// TIA Portal V21 export
FUNCTION "FC601" : Void   // FC601, LAD
TITLE = FC601
{ S7_Optimized_Access := 'TRUE' }
// MAIN CIP CALL BLOCK
// stored: AutoNumber false, SetENOAutomatically false
   VAR_TEMP   // added for the SCL form of the ladder/FBD networks
      _w1 : Bool;
      _w2 : Bool;
      _w3 : Bool;
   END_VAR
BEGIN

REGION Network 1: "FC604"
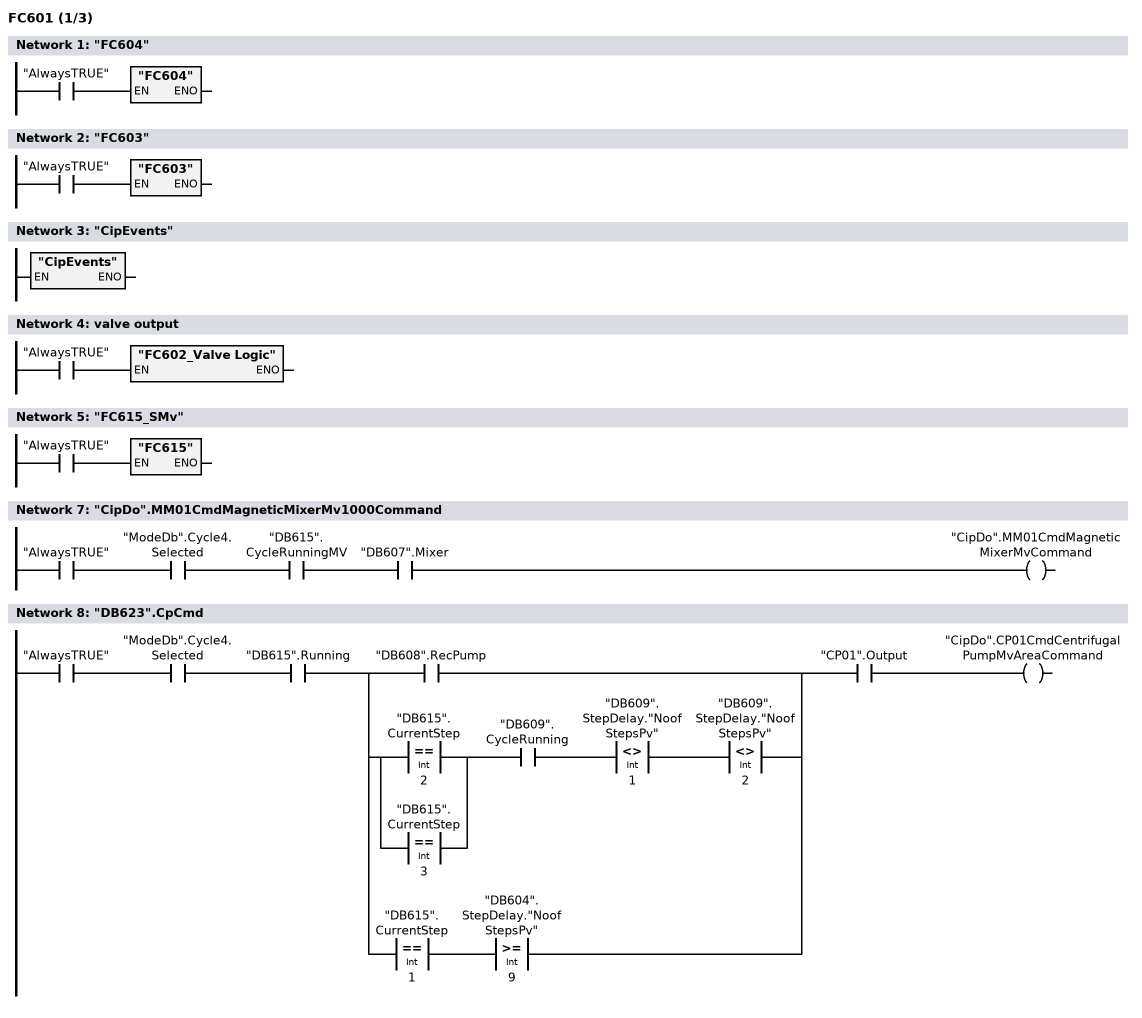
   RUNG wire#powerrail
      Contact( "AlwaysTRUE" )
      "FC604"()
   END_RUNG
   // the same network as SCL:
   IF "AlwaysTRUE" THEN "FC604"(); END_IF;
END_REGION

REGION Network 2: "FC603"
   RUNG wire#powerrail
      Contact( "AlwaysTRUE" )
      "FC603"()
   END_RUNG
   // the same network as SCL:
   IF "AlwaysTRUE" THEN "FC603"(); END_IF;
END_REGION

REGION Network 3: "CipEvents"
   RUNG wire#powerrail
      "CipEvents"()
   END_RUNG
   // the same network as SCL:
   "CipEvents"();
END_REGION

REGION Network 4: valve output
   RUNG wire#powerrail
      Contact( "AlwaysTRUE" )
      "FC602_Valve Logic"()
   END_RUNG
   // the same network as SCL:
   IF "AlwaysTRUE" THEN "FC602_Valve Logic"(); END_IF;
END_REGION

REGION Network 5: "FC615_SMv"
   RUNG wire#powerrail
      Contact( "AlwaysTRUE" )
      "FC615"()
   END_RUNG
   // the same network as SCL:
   IF "AlwaysTRUE" THEN "FC615"(); END_IF;
END_REGION

REGION Network 6: *************DO ***********************
END_REGION

REGION Network 7: "CipDo".MM01CmdMagneticMixerMv1000Command
   RUNG wire#powerrail
      Contact( "AlwaysTRUE" )
      Contact( "ModeDb".Cycle4.Selected )
      Contact( "DB615".CycleRunningMV )
      Contact( "DB607".Mixer )
      Coil( "CipDo".MM01CmdMagneticMixerMvCommand )
   END_RUNG
   // the same network as SCL:
   "CipDo".MM01CmdMagneticMixerMvCommand := "AlwaysTRUE" AND "ModeDb".Cycle4.Selected AND "DB615".CycleRunningMV AND "DB607".Mixer;
END_REGION

REGION Network 8: "DB623".CpCmd
   RUNG wire#powerrail
      Contact( "AlwaysTRUE" )
      Contact( "ModeDb".Cycle4.Selected )
      Contact( "DB615".Running )
      wire#w1
      Contact( "DB608".RecPump )
      wire#w2
      Contact( "CP01".Output )
      Coil( "CipDo".CP01CmdCentrifugalPumpMvAreaCommand )
   END_RUNG
   RUNG wire#w1
      { S7_Templates := "SrcType := Int" } EQ_Contact(in1 := "DB615".CurrentStep, in2 := 2)
      wire#w3
      Contact( "DB609".CycleRunning )
      { S7_Templates := "SrcType := Int" } NE_Contact(in1 := "DB609".StepDelay."Noof StepsPv", in2 := 1)
      { S7_Templates := "SrcType := Int" } NE_Contact(in1 := "DB609".StepDelay."Noof StepsPv", in2 := 2)
   END_RUNG wire#w2
   RUNG wire#w1
      { S7_Templates := "SrcType := Int" } EQ_Contact(in1 := "DB615".CurrentStep, in2 := 3)
   END_RUNG wire#w3
   RUNG wire#w1
      { S7_Templates := "SrcType := Int" } EQ_Contact(in1 := "DB615".CurrentStep, in2 := 1)
      { S7_Templates := "SrcType := Int" } GE_Contact(in1 := "DB604".StepDelay."Noof StepsPv", in2 := 9)
   END_RUNG wire#w2
   // the same network as SCL:
   "CipDo".CP01CmdCentrifugalPumpMvAreaCommand := "AlwaysTRUE" AND "ModeDb".Cycle4.Selected AND "DB615".Running AND ("DB608".RecPump OR ((("DB615".CurrentStep = 2) OR ("DB615".CurrentStep = 3)) AND "DB609".CycleRunning AND ("DB609".StepDelay."Noof StepsPv" <> 1) AND ("DB609".StepDelay."Noof StepsPv" <> 2)) OR (("DB615".CurrentStep = 1) AND ("DB604".StepDelay."Noof StepsPv" >= 9))) AND "CP01".Output;
END_REGION

REGION Network 9: "CipDo".CP01CmdCentrifugalPump
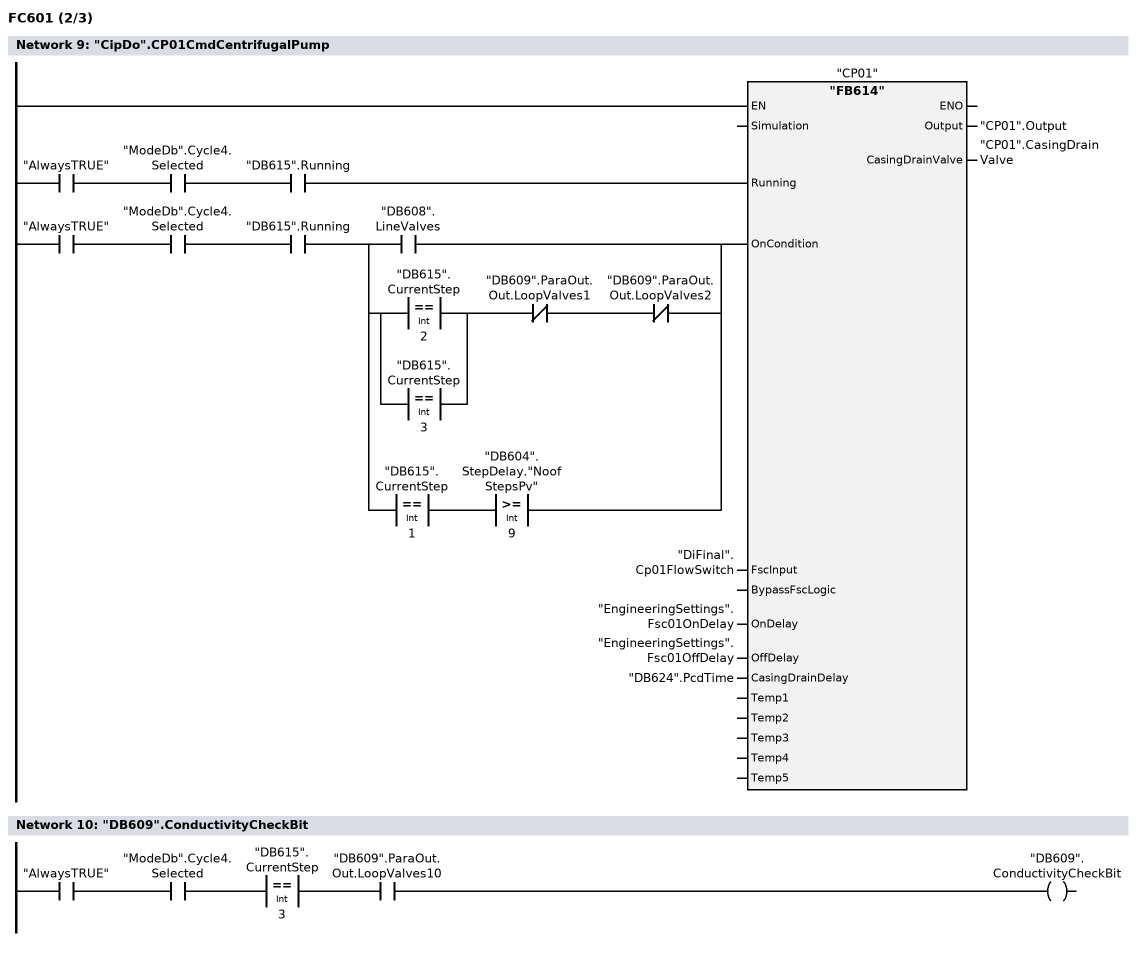
   RUNG wire#powerrail
      "CP01"(Running := wire#w1, OnCondition := wire#w4, Simulation :=, FscInput := "DiFinal".Cp01FlowSwitch, BypassFscLogic :=, OnDelay := "EngineeringSettings".Fsc01OnDelay, OffDelay := "EngineeringSettings".Fsc01OffDelay, CasingDrainDelay := "DB624".PcdTime, Temp1 :=, Temp2 :=, Temp3 :=, Temp4 :=, Temp5 :=, Output => "CP01".Output, CasingDrainValve => "CP01".CasingDrainValve)
   END_RUNG
   RUNG wire#powerrail
      Contact( "AlwaysTRUE" )
      Contact( "ModeDb".Cycle4.Selected )
      Contact( "DB615".Running )
   END_RUNG wire#w1
   RUNG wire#powerrail
      Contact( "AlwaysTRUE" )
      Contact( "ModeDb".Cycle4.Selected )
      Contact( "DB615".Running )
      wire#w2
      Contact( "DB608".LineValves )
   END_RUNG wire#w4
   RUNG wire#w2
      { S7_Templates := "SrcType := Int" } EQ_Contact(in1 := "DB615".CurrentStep, in2 := 2)
      wire#w3
      I_Contact( "DB609".ParaOut.Out.LoopValves1 )
      I_Contact( "DB609".ParaOut.Out.LoopValves2 )
   END_RUNG wire#w4
   RUNG wire#w2
      { S7_Templates := "SrcType := Int" } EQ_Contact(in1 := "DB615".CurrentStep, in2 := 3)
   END_RUNG wire#w3
   RUNG wire#w2
      { S7_Templates := "SrcType := Int" } EQ_Contact(in1 := "DB615".CurrentStep, in2 := 1)
      { S7_Templates := "SrcType := Int" } GE_Contact(in1 := "DB604".StepDelay."Noof StepsPv", in2 := 9)
   END_RUNG wire#w4
   // the same network as SCL:
   "CP01"(Running := "AlwaysTRUE" AND "ModeDb".Cycle4.Selected AND "DB615".Running,   // "FB614"
          OnCondition := "AlwaysTRUE" AND "ModeDb".Cycle4.Selected AND "DB615".Running AND ("DB608".LineValves OR ((("DB615".CurrentStep = 2) OR ("DB615".CurrentStep = 3)) AND NOT "DB609".ParaOut.Out.LoopValves1 AND NOT "DB609".ParaOut.Out.LoopValves2) OR (("DB615".CurrentStep = 1) AND ("DB604".StepDelay."Noof StepsPv" >= 9))),
          FscInput := "DiFinal".Cp01FlowSwitch,
          OnDelay := "EngineeringSettings".Fsc01OnDelay,
          OffDelay := "EngineeringSettings".Fsc01OffDelay,
          CasingDrainDelay := "DB624".PcdTime,
          Output => "CP01".Output,
          CasingDrainValve => "CP01".CasingDrainValve);
END_REGION

REGION Network 10: "DB609".ConductivityCheckBit
   RUNG wire#powerrail
      Contact( "AlwaysTRUE" )
      Contact( "ModeDb".Cycle4.Selected )
      { S7_Templates := "SrcType := Int" } EQ_Contact(in1 := "DB615".CurrentStep, in2 := 3)
      Contact( "DB609".ParaOut.Out.LoopValves10 )
      Coil( "DB609".ConductivityCheckBit )
   END_RUNG
   // the same network as SCL:
   "DB609".ConductivityCheckBit := "AlwaysTRUE" AND "ModeDb".Cycle4.Selected AND ("DB615".CurrentStep = 3) AND "DB609".ParaOut.Out.LoopValves10;
END_REGION

REGION Network 12: "ProcessAlarms".MvVesselWfiFlowLow
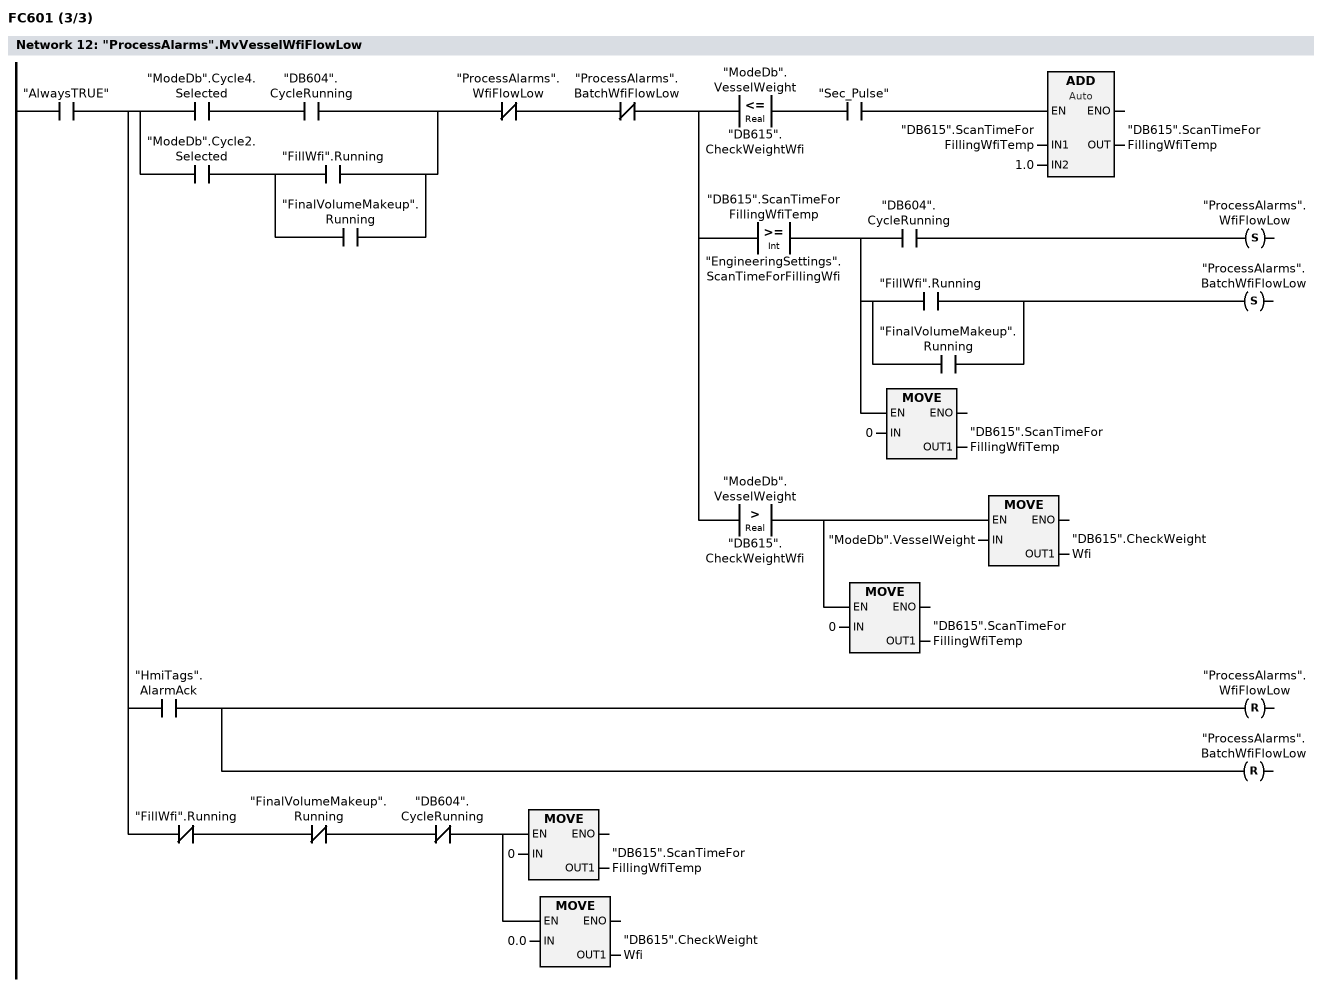
   RUNG wire#powerrail
      Contact( "AlwaysTRUE" )
      wire#w1
      Contact( "ModeDb".Cycle4.Selected )
      Contact( "DB604".CycleRunning )
      wire#w2
      I_Contact( "ProcessAlarms".WfiFlowLow )
      I_Contact( "ProcessAlarms".BatchWfiFlowLow )
      wire#w4
      { S7_Templates := "SrcType := Real" } LE_Contact(in1 := "ModeDb".VesselWeight, in2 := "DB615".CheckWeightWfi)
      Contact( "Sec_Pulse" )
      Add(in1 := "DB615".ScanTimeForFillingWfiTemp, in2 := 1.0, out => "DB615".ScanTimeForFillingWfiTemp)
   END_RUNG
   RUNG wire#w1
      Contact( "ModeDb".Cycle2.Selected )
      wire#w3
      Contact( "FillWfi".Running )
   END_RUNG wire#w2
   RUNG wire#w3
      Contact( "FinalVolumeMakeup".Running )
   END_RUNG wire#w2
   RUNG wire#w4
      { S7_Templates := "SrcType := Int" } GE_Contact(in1 := "DB615".ScanTimeForFillingWfiTemp, in2 := "EngineeringSettings".ScanTimeForFillingWfi)
      wire#w5
      Contact( "DB604".CycleRunning )
      S_Coil( "ProcessAlarms".WfiFlowLow )
   END_RUNG
   RUNG wire#w5
      Contact( "FillWfi".Running )
      wire#w6
      S_Coil( "ProcessAlarms".BatchWfiFlowLow )
   END_RUNG
   RUNG wire#w5
      Contact( "FinalVolumeMakeup".Running )
   END_RUNG wire#w6
   RUNG wire#w5
      Move(in := 0, out1 => "DB615".ScanTimeForFillingWfiTemp)
   END_RUNG
   RUNG wire#w4
      { S7_Templates := "SrcType := Real" } GT_Contact(in1 := "ModeDb".VesselWeight, in2 := "DB615".CheckWeightWfi)
      wire#w7
      Move(in := "ModeDb".VesselWeight, out1 => "DB615".CheckWeightWfi)
   END_RUNG
   RUNG wire#w7
      Move(in := 0, out1 => "DB615".ScanTimeForFillingWfiTemp)
   END_RUNG
   RUNG wire#w1
      Contact( "HmiTags".AlarmAck )
      wire#w8
      R_Coil( "ProcessAlarms".WfiFlowLow )
   END_RUNG
   RUNG wire#w8
      R_Coil( "ProcessAlarms".BatchWfiFlowLow )
   END_RUNG
   RUNG wire#w1
      I_Contact( "FillWfi".Running )
      I_Contact( "FinalVolumeMakeup".Running )
      I_Contact( "DB604".CycleRunning )
      wire#w9
      Move(in := 0, out1 => "DB615".ScanTimeForFillingWfiTemp)
   END_RUNG
   RUNG wire#w9
      Move(in := 0.0, out1 => "DB615".CheckWeightWfi)
   END_RUNG
   // the same network as SCL:
   #_w1 := "AlwaysTRUE" AND (("ModeDb".Cycle4.Selected AND "DB604".CycleRunning) OR ("ModeDb".Cycle2.Selected AND ("FillWfi".Running OR "FinalVolumeMakeup".Running))) AND NOT "ProcessAlarms".WfiFlowLow AND NOT "ProcessAlarms".BatchWfiFlowLow;
   IF #_w1 AND ("ModeDb".VesselWeight <= "DB615".CheckWeightWfi) AND "Sec_Pulse" THEN
       "DB615".ScanTimeForFillingWfiTemp := "DB615".ScanTimeForFillingWfiTemp + 1.0;
   END_IF;
   #_w2 := #_w1 AND ("DB615".ScanTimeForFillingWfiTemp >= "EngineeringSettings".ScanTimeForFillingWfi);
   IF #_w2 AND "DB604".CycleRunning THEN "ProcessAlarms".WfiFlowLow := TRUE; END_IF;
   IF #_w2 AND ("FillWfi".Running OR "FinalVolumeMakeup".Running) THEN
       "ProcessAlarms".BatchWfiFlowLow := TRUE;
   END_IF;
   IF #_w2 THEN "DB615".ScanTimeForFillingWfiTemp := 0; END_IF;
   #_w3 := #_w1 AND ("ModeDb".VesselWeight > "DB615".CheckWeightWfi);
   IF #_w3 THEN
       "DB615".CheckWeightWfi := "ModeDb".VesselWeight;
       "DB615".ScanTimeForFillingWfiTemp := 0;
   END_IF;
   IF "AlwaysTRUE" AND "HmiTags".AlarmAck THEN
       "ProcessAlarms".WfiFlowLow := FALSE;
       "ProcessAlarms".BatchWfiFlowLow := FALSE;
   END_IF;
   IF "AlwaysTRUE" AND NOT "FillWfi".Running AND NOT "FinalVolumeMakeup".Running AND NOT "DB604".CycleRunning THEN
       "DB615".ScanTimeForFillingWfiTemp := 0;
       "DB615".CheckWeightWfi := 0.0;
   END_IF;
END_REGION
END_FUNCTION
